RoboDK station: Simulation.rdk

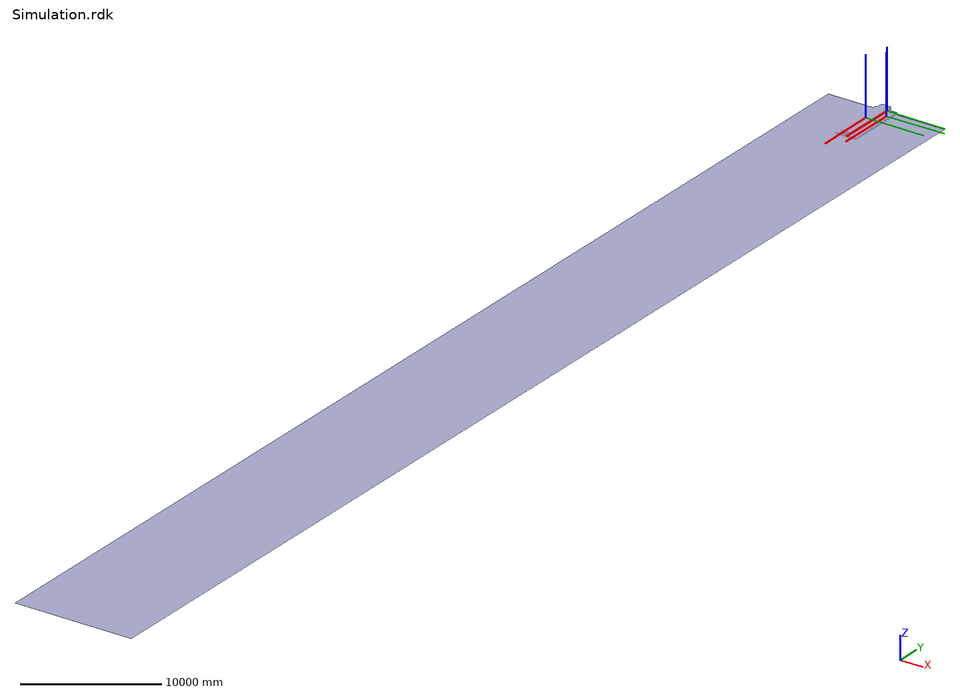
[picture v0: the station drawn from its stored meshes, robots at their saved joint values, targets as dots, program paths as lines]
Station Simulation (saved by RoboDK 5.2.5). Poses are relative to the parent item; angles as X-Y-Z fixed-axis rotations.
  - object Floor at (0, -50000, 0) mm, size 10000 x 100000 x 5 mm, geometry from Floor.stp
  - frame Conveyor Belt Wide (2m) Base at (0, 0, -365.24) mm, rotated rx 0 ry 0 rz -90 deg
    - robot Conveyor Belt Wide (2m): 1 axes
        modified DH rows (alpha deg, a mm, theta deg, d mm): 0, 0, 0, 0 linear
        base shift (0, 0, 0) mm, rotated rx 0 ry 90 rz 0 deg
        joint limits [-900000] to [900000]; home [0]; saved at [-79.153]
      - frame Carriage at (0, 0, 0) mm
        - object Support at (2600, 0, 0) mm, rotated rx 0 ry 0 rz 90 deg, size 1800 x 5000 x 500 mm, geometry from Support.stp
        - frame Car_Base at (2600, 0, 500) mm
